// TIA Portal V17 export
// export: Created 2025-03-07T09:16:32.9200456Z, ExportSetting WithDefaults, DisplayName Totally Integrated Automation Portal, DisplayVersion V17 Update 8, DisplayName TIA Portal Openness, DisplayVersion V17 Update 8, DisplayName TIA Portal Version Control Interface, DisplayVersion V17, DisplayName SINAMICS Startdrive Advanced, DisplayVersion V17 SP2, DisplayName SINAMICS Startdrive G110M, G120, G120C, G120D, G120P, G115D, DisplayVersion V17 SP2, DisplayName SINAMICS Startdrive G130, G150, S120, S150, SINAMICS MV, S210, DisplayVersion V17 SP2, DisplayName STEP 7 Professional, DisplayVersion V17 Update 8, DisplayName SINUMERIK ONE STEP 7 Toolbox, DisplayVersion V17 Update 12, DisplayName SINUMERIK 840D sl STEP 7 Toolbox, DisplayVersion V17 Update 12, DisplayName STEP 7 Safety, DisplayVersion V17 Update 6, DisplayName WinCC Advanced, DisplayVersion V17 Update 8
DATA_BLOCK "LBP_SpindleTempSensor"   // DB1002
TITLE = Spindle temperature sensors / Sensores de temperatura del cabezal / Spindeltemperatursensoren
{ S7_Optimized_Access := 'FALSE'; DB_Accessible_From_OPC_UA := 'FALSE' }
AUTHOR : SINUMERIK
FAMILY : SINUMERIK_ONE
VERSION : 6.15
// Interface between user program and operating software, contains signals for spindle temperature sensors / La interfaz entre programa de usuario y software operativo contiene señales para sensores de temperatura del cabezal / Schnittstelle zwischen Anwenderprogramm und Betriebssoftware, enthält Signale für Spindeltemperatursensoren
// stored: AutoNumber false, DBAccessibleFromOPCUA false, DBAccessibleFromWebserver true, IsOnlyStoredInLoadMemory false, IsWriteProtectedInAS false
   VAR RETAIN
      Sp : Array[1..2] of Struct   // Spindel / Spindle / Cabezal
         TS : Array[1..6] of Struct   // Temperatursensor / Temperature sensor / Sensor de temperatura
            MountPlace : Int;   // Platz der Sensorbaugruppe / Sensor assembly location / Ubicación del conjunto de sensores
            Res1 : Int;
            ActVal : Real;   // Temperatursensor Istwert [°C] / Temperature sensor actual value [°C] / Sensor de temperatura valor real [°C]
            WarnThreshold : Real;   // Temperatursensor Warnschwellwert / Temperature sensor warning threshold value [°C] / Sensor de temperatura umbral de alarma
            WarnNumLimitViol : Int;   // Anzahl der Warnschwellwert-Verletzungen / Number of warning threshold value violations / Número de vulneraciones del umbral de alarma
            WarnTsViolYY : Byte;   // Letzte Warnschwellwert-Verletzung: Jahr / Last warning threshold value violation: year / Última vulneración del umbral de alarma: año
            WarnTsViolMM : Byte;   // Letzte Warnschwellwert-Verletzung: Monat / Last warning threshold value violation: month / Última vulneración del umbral de alarma: mes
            WarnTsViolDD : Byte;   // Letzte Warnschwellwert-Verletzung: Tag / Last warning threshold value violation: day / Última vulneración del umbral de fallo: día
            WarnTsViolH : Byte;   // Letzte Warnschwellwert-Verletzung: Stunde / Last warning threshold value violation: hour / Última vulneración del umbral de fallo: hora
            WarnTsViolM : Byte;   // Letzte Warnschwellwert-Verletzung: Minute / Last warning threshold value violation: minute / Última vulneración del umbral de fallo: minuto
            WarnTsViolS : Byte;   // Letzte Warnschwellwert-Verletzung: Sekunde / Last warning threshold value violation: second / Última vulneración del umbral de alarma: segundo
            WarnDurLimitViol : DInt;   // Dauer der Warnschwellwert-Verletzungen / Duration of warning threshold value violations / Duración de vulneraciones del umbral de alarma
            FaultThreshold : Real;   // Temperatursensor Fehlerschwellwert / Temperature sensor fault threshold value [°C] / Sensor de temperatura umbral de fallo
            FaultNumLimitViol : Int;   // Anzahl der Fehlerschwellwert-Verletzungen / Number of fault threshold value violations / Número de vulneraciones del umbral de fallo
            FaultTsViolYY : Byte;   // Letzte Fehlerschwellwert-Verletzung: Jahr / Last fault threshold value violation: year / Última vulneración del umbral de fallo: año
            FaultTsViolMM : Byte;   // Letzte Fehlerschwellwert-Verletzung: Monat / Last fault threshold value violation: month / Última vulneración del umbral de fallo: mes
            FaultTsViolDD : Byte;   // Letzte Fehlerschwellwert-Verletzung: Tag / Last fault threshold value violation: day / Última vulneración del umbral de fallo: día
            FaultTsViolH : Byte;   // Letzte Fehlerschwellwert-Verletzung: Stunde / Last fault threshold value violation: hour / Última vulneración del umbral de fallo: hora
            FaultTsViolM : Byte;   // Letzte Fehlerschwellwert-Verletzung: Minute / Last fault threshold value violation: minute / Última vulneración del umbral de fallo: minuto
            FaultTsViolS : Byte;   // Letzte Fehlerschwellwert-Verletzung: Sekunde / Last fault threshold value violation: second / Última vulneración del umbral de fallo: segundo
            FaultDurLimitViol : DInt;   // Dauer der Fehlerschwellwert-Verletzungen / Duration of fault threshold value violations / Duración de vulneraciones del umbral de fallo
         END_STRUCT;
      END_STRUCT;
   END_VAR
BEGIN
   // Sp[1].TS[2].MountPlace : Platz der Sensorbaugruppe / Sensor assembly location / Ubicación del conjunto de sensores
   // Sp[1].TS[3].MountPlace : Platz der Sensorbaugruppe / Sensor assembly location / Ubicación del conjunto de sensores
   // Sp[1].TS[4].MountPlace : Platz der Sensorbaugruppe / Sensor assembly location / Ubicación del conjunto de sensores
   // Sp[1].TS[5].MountPlace : Platz der Sensorbaugruppe / Sensor assembly location / Ubicación del conjunto de sensores
   // Sp[1].TS[6].MountPlace : Platz der Sensorbaugruppe / Sensor assembly location / Ubicación del conjunto de sensores
   // Sp[2].TS[1].MountPlace : Platz der Sensorbaugruppe / Sensor assembly location / Ubicación del conjunto de sensores
   // Sp[2].TS[2].MountPlace : Platz der Sensorbaugruppe / Sensor assembly location / Ubicación del conjunto de sensores
   // Sp[2].TS[3].MountPlace : Platz der Sensorbaugruppe / Sensor assembly location / Ubicación del conjunto de sensores
   // Sp[2].TS[4].MountPlace : Platz der Sensorbaugruppe / Sensor assembly location / Ubicación del conjunto de sensores
   // Sp[2].TS[5].MountPlace : Platz der Sensorbaugruppe / Sensor assembly location / Ubicación del conjunto de sensores
   // Sp[2].TS[6].MountPlace : Platz der Sensorbaugruppe / Sensor assembly location / Ubicación del conjunto de sensores
   // Sp[1].TS[2].ActVal : Temperatursensor Istwert [°C] / Temperature sensor actual value [°C] / Sensor de temperatura valor real [°C]
   // Sp[1].TS[3].ActVal : Temperatursensor Istwert [°C] / Temperature sensor actual value [°C] / Sensor de temperatura valor real [°C]
   // Sp[1].TS[4].ActVal : Temperatursensor Istwert [°C] / Temperature sensor actual value [°C] / Sensor de temperatura valor real [°C]
   // Sp[1].TS[5].ActVal : Temperatursensor Istwert [°C] / Temperature sensor actual value [°C] / Sensor de temperatura valor real [°C]
   // Sp[1].TS[6].ActVal : Temperatursensor Istwert [°C] / Temperature sensor actual value [°C] / Sensor de temperatura valor real [°C]
   // Sp[2].TS[1].ActVal : Temperatursensor Istwert [°C] / Temperature sensor actual value [°C] / Sensor de temperatura valor real [°C]
   // Sp[2].TS[2].ActVal : Temperatursensor Istwert [°C] / Temperature sensor actual value [°C] / Sensor de temperatura valor real [°C]
   // Sp[2].TS[3].ActVal : Temperatursensor Istwert [°C] / Temperature sensor actual value [°C] / Sensor de temperatura valor real [°C]
   // Sp[2].TS[4].ActVal : Temperatursensor Istwert [°C] / Temperature sensor actual value [°C] / Sensor de temperatura valor real [°C]
   // Sp[2].TS[5].ActVal : Temperatursensor Istwert [°C] / Temperature sensor actual value [°C] / Sensor de temperatura valor real [°C]
   // Sp[2].TS[6].ActVal : Temperatursensor Istwert [°C] / Temperature sensor actual value [°C] / Sensor de temperatura valor real [°C]
   // Sp[1].TS[2].WarnThreshold : Temperatursensor Warnschwellwert / Temperature sensor warning threshold value [°C] / Sensor de temperatura umbral de alarma
   // Sp[1].TS[3].WarnThreshold : Temperatursensor Warnschwellwert / Temperature sensor warning threshold value [°C] / Sensor de temperatura umbral de alarma
   // Sp[1].TS[4].WarnThreshold : Temperatursensor Warnschwellwert / Temperature sensor warning threshold value [°C] / Sensor de temperatura umbral de alarma
   // Sp[1].TS[5].WarnThreshold : Temperatursensor Warnschwellwert / Temperature sensor warning threshold value [°C] / Sensor de temperatura umbral de alarma
   // Sp[1].TS[6].WarnThreshold : Temperatursensor Warnschwellwert / Temperature sensor warning threshold value [°C] / Sensor de temperatura umbral de alarma
   // Sp[2].TS[1].WarnThreshold : Temperatursensor Warnschwellwert / Temperature sensor warning threshold value [°C] / Sensor de temperatura umbral de alarma
   // Sp[2].TS[2].WarnThreshold : Temperatursensor Warnschwellwert / Temperature sensor warning threshold value [°C] / Sensor de temperatura umbral de alarma
   // Sp[2].TS[3].WarnThreshold : Temperatursensor Warnschwellwert / Temperature sensor warning threshold value [°C] / Sensor de temperatura umbral de alarma
   // Sp[2].TS[4].WarnThreshold : Temperatursensor Warnschwellwert / Temperature sensor warning threshold value [°C] / Sensor de temperatura umbral de alarma
   // Sp[2].TS[5].WarnThreshold : Temperatursensor Warnschwellwert / Temperature sensor warning threshold value [°C] / Sensor de temperatura umbral de alarma
   // Sp[2].TS[6].WarnThreshold : Temperatursensor Warnschwellwert / Temperature sensor warning threshold value [°C] / Sensor de temperatura umbral de alarma
   // Sp[1].TS[2].WarnNumLimitViol : Anzahl der Warnschwellwert-Verletzungen / Number of warning threshold value violations / Número de vulneraciones del umbral de alarma
   // Sp[1].TS[3].WarnNumLimitViol : Anzahl der Warnschwellwert-Verletzungen / Number of warning threshold value violations / Número de vulneraciones del umbral de alarma
   // Sp[1].TS[4].WarnNumLimitViol : Anzahl der Warnschwellwert-Verletzungen / Number of warning threshold value violations / Número de vulneraciones del umbral de alarma
   // Sp[1].TS[5].WarnNumLimitViol : Anzahl der Warnschwellwert-Verletzungen / Number of warning threshold value violations / Número de vulneraciones del umbral de alarma
   // Sp[1].TS[6].WarnNumLimitViol : Anzahl der Warnschwellwert-Verletzungen / Number of warning threshold value violations / Número de vulneraciones del umbral de alarma
   // Sp[2].TS[1].WarnNumLimitViol : Anzahl der Warnschwellwert-Verletzungen / Number of warning threshold value violations / Número de vulneraciones del umbral de alarma
   // Sp[2].TS[2].WarnNumLimitViol : Anzahl der Warnschwellwert-Verletzungen / Number of warning threshold value violations / Número de vulneraciones del umbral de alarma
   // Sp[2].TS[3].WarnNumLimitViol : Anzahl der Warnschwellwert-Verletzungen / Number of warning threshold value violations / Número de vulneraciones del umbral de alarma
   // Sp[2].TS[4].WarnNumLimitViol : Anzahl der Warnschwellwert-Verletzungen / Number of warning threshold value violations / Número de vulneraciones del umbral de alarma
   // Sp[2].TS[5].WarnNumLimitViol : Anzahl der Warnschwellwert-Verletzungen / Number of warning threshold value violations / Número de vulneraciones del umbral de alarma
   // Sp[2].TS[6].WarnNumLimitViol : Anzahl der Warnschwellwert-Verletzungen / Number of warning threshold value violations / Número de vulneraciones del umbral de alarma
   // Sp[1].TS[2].WarnTsViolYY : Letzte Warnschwellwert-Verletzung: Jahr / Last warning threshold value violation: year / Última vulneración del umbral de alarma: año
   // Sp[1].TS[3].WarnTsViolYY : Letzte Warnschwellwert-Verletzung: Jahr / Last warning threshold value violation: year / Última vulneración del umbral de alarma: año
   // Sp[1].TS[4].WarnTsViolYY : Letzte Warnschwellwert-Verletzung: Jahr / Last warning threshold value violation: year / Última vulneración del umbral de alarma: año
   // Sp[1].TS[5].WarnTsViolYY : Letzte Warnschwellwert-Verletzung: Jahr / Last warning threshold value violation: year / Última vulneración del umbral de alarma: año
   // Sp[1].TS[6].WarnTsViolYY : Letzte Warnschwellwert-Verletzung: Jahr / Last warning threshold value violation: year / Última vulneración del umbral de alarma: año
   // Sp[2].TS[1].WarnTsViolYY : Letzte Warnschwellwert-Verletzung: Jahr / Last warning threshold value violation: year / Última vulneración del umbral de alarma: año
   // Sp[2].TS[2].WarnTsViolYY : Letzte Warnschwellwert-Verletzung: Jahr / Last warning threshold value violation: year / Última vulneración del umbral de alarma: año
   // Sp[2].TS[3].WarnTsViolYY : Letzte Warnschwellwert-Verletzung: Jahr / Last warning threshold value violation: year / Última vulneración del umbral de alarma: año
   // Sp[2].TS[4].WarnTsViolYY : Letzte Warnschwellwert-Verletzung: Jahr / Last warning threshold value violation: year / Última vulneración del umbral de alarma: año
   // Sp[2].TS[5].WarnTsViolYY : Letzte Warnschwellwert-Verletzung: Jahr / Last warning threshold value violation: year / Última vulneración del umbral de alarma: año
   // Sp[2].TS[6].WarnTsViolYY : Letzte Warnschwellwert-Verletzung: Jahr / Last warning threshold value violation: year / Última vulneración del umbral de alarma: año
   // Sp[1].TS[2].WarnTsViolMM : Letzte Warnschwellwert-Verletzung: Monat / Last warning threshold value violation: month / Última vulneración del umbral de alarma: mes
   // Sp[1].TS[3].WarnTsViolMM : Letzte Warnschwellwert-Verletzung: Monat / Last warning threshold value violation: month / Última vulneración del umbral de alarma: mes
   // Sp[1].TS[4].WarnTsViolMM : Letzte Warnschwellwert-Verletzung: Monat / Last warning threshold value violation: month / Última vulneración del umbral de alarma: mes
   // Sp[1].TS[5].WarnTsViolMM : Letzte Warnschwellwert-Verletzung: Monat / Last warning threshold value violation: month / Última vulneración del umbral de alarma: mes
   // Sp[1].TS[6].WarnTsViolMM : Letzte Warnschwellwert-Verletzung: Monat / Last warning threshold value violation: month / Última vulneración del umbral de alarma: mes
   // Sp[2].TS[1].WarnTsViolMM : Letzte Warnschwellwert-Verletzung: Monat / Last warning threshold value violation: month / Última vulneración del umbral de alarma: mes
   // Sp[2].TS[2].WarnTsViolMM : Letzte Warnschwellwert-Verletzung: Monat / Last warning threshold value violation: month / Última vulneración del umbral de alarma: mes
   // Sp[2].TS[3].WarnTsViolMM : Letzte Warnschwellwert-Verletzung: Monat / Last warning threshold value violation: month / Última vulneración del umbral de alarma: mes
   // Sp[2].TS[4].WarnTsViolMM : Letzte Warnschwellwert-Verletzung: Monat / Last warning threshold value violation: month / Última vulneración del umbral de alarma: mes
   // Sp[2].TS[5].WarnTsViolMM : Letzte Warnschwellwert-Verletzung: Monat / Last warning threshold value violation: month / Última vulneración del umbral de alarma: mes
   // Sp[2].TS[6].WarnTsViolMM : Letzte Warnschwellwert-Verletzung: Monat / Last warning threshold value violation: month / Última vulneración del umbral de alarma: mes
   // Sp[1].TS[2].WarnTsViolDD : Letzte Warnschwellwert-Verletzung: Tag / Last warning threshold value violation: day / Última vulneración del umbral de fallo: día
   // Sp[1].TS[3].WarnTsViolDD : Letzte Warnschwellwert-Verletzung: Tag / Last warning threshold value violation: day / Última vulneración del umbral de fallo: día
   // Sp[1].TS[4].WarnTsViolDD : Letzte Warnschwellwert-Verletzung: Tag / Last warning threshold value violation: day / Última vulneración del umbral de fallo: día
   // Sp[1].TS[5].WarnTsViolDD : Letzte Warnschwellwert-Verletzung: Tag / Last warning threshold value violation: day / Última vulneración del umbral de fallo: día
   // Sp[1].TS[6].WarnTsViolDD : Letzte Warnschwellwert-Verletzung: Tag / Last warning threshold value violation: day / Última vulneración del umbral de fallo: día
   // Sp[2].TS[1].WarnTsViolDD : Letzte Warnschwellwert-Verletzung: Tag / Last warning threshold value violation: day / Última vulneración del umbral de fallo: día
   // Sp[2].TS[2].WarnTsViolDD : Letzte Warnschwellwert-Verletzung: Tag / Last warning threshold value violation: day / Última vulneración del umbral de fallo: día
   // Sp[2].TS[3].WarnTsViolDD : Letzte Warnschwellwert-Verletzung: Tag / Last warning threshold value violation: day / Última vulneración del umbral de fallo: día
   // Sp[2].TS[4].WarnTsViolDD : Letzte Warnschwellwert-Verletzung: Tag / Last warning threshold value violation: day / Última vulneración del umbral de fallo: día
   // Sp[2].TS[5].WarnTsViolDD : Letzte Warnschwellwert-Verletzung: Tag / Last warning threshold value violation: day / Última vulneración del umbral de fallo: día
   // Sp[2].TS[6].WarnTsViolDD : Letzte Warnschwellwert-Verletzung: Tag / Last warning threshold value violation: day / Última vulneración del umbral de fallo: día
   // Sp[1].TS[2].WarnTsViolH : Letzte Warnschwellwert-Verletzung: Stunde / Last warning threshold value violation: hour / Última vulneración del umbral de fallo: hora
   // Sp[1].TS[3].WarnTsViolH : Letzte Warnschwellwert-Verletzung: Stunde / Last warning threshold value violation: hour / Última vulneración del umbral de fallo: hora
   // Sp[1].TS[4].WarnTsViolH : Letzte Warnschwellwert-Verletzung: Stunde / Last warning threshold value violation: hour / Última vulneración del umbral de fallo: hora
   // Sp[1].TS[5].WarnTsViolH : Letzte Warnschwellwert-Verletzung: Stunde / Last warning threshold value violation: hour / Última vulneración del umbral de fallo: hora
   // Sp[1].TS[6].WarnTsViolH : Letzte Warnschwellwert-Verletzung: Stunde / Last warning threshold value violation: hour / Última vulneración del umbral de fallo: hora
   // Sp[2].TS[1].WarnTsViolH : Letzte Warnschwellwert-Verletzung: Stunde / Last warning threshold value violation: hour / Última vulneración del umbral de fallo: hora
   // Sp[2].TS[2].WarnTsViolH : Letzte Warnschwellwert-Verletzung: Stunde / Last warning threshold value violation: hour / Última vulneración del umbral de fallo: hora
   // Sp[2].TS[3].WarnTsViolH : Letzte Warnschwellwert-Verletzung: Stunde / Last warning threshold value violation: hour / Última vulneración del umbral de fallo: hora
   // Sp[2].TS[4].WarnTsViolH : Letzte Warnschwellwert-Verletzung: Stunde / Last warning threshold value violation: hour / Última vulneración del umbral de fallo: hora
   // Sp[2].TS[5].WarnTsViolH : Letzte Warnschwellwert-Verletzung: Stunde / Last warning threshold value violation: hour / Última vulneración del umbral de fallo: hora
   // Sp[2].TS[6].WarnTsViolH : Letzte Warnschwellwert-Verletzung: Stunde / Last warning threshold value violation: hour / Última vulneración del umbral de fallo: hora
   // Sp[1].TS[2].WarnTsViolM : Letzte Warnschwellwert-Verletzung: Minute / Last warning threshold value violation: minute / Última vulneración del umbral de fallo: minuto
   // Sp[1].TS[3].WarnTsViolM : Letzte Warnschwellwert-Verletzung: Minute / Last warning threshold value violation: minute / Última vulneración del umbral de fallo: minuto
   // Sp[1].TS[4].WarnTsViolM : Letzte Warnschwellwert-Verletzung: Minute / Last warning threshold value violation: minute / Última vulneración del umbral de fallo: minuto
   // Sp[1].TS[5].WarnTsViolM : Letzte Warnschwellwert-Verletzung: Minute / Last warning threshold value violation: minute / Última vulneración del umbral de fallo: minuto
   // Sp[1].TS[6].WarnTsViolM : Letzte Warnschwellwert-Verletzung: Minute / Last warning threshold value violation: minute / Última vulneración del umbral de fallo: minuto
   // Sp[2].TS[1].WarnTsViolM : Letzte Warnschwellwert-Verletzung: Minute / Last warning threshold value violation: minute / Última vulneración del umbral de fallo: minuto
   // Sp[2].TS[2].WarnTsViolM : Letzte Warnschwellwert-Verletzung: Minute / Last warning threshold value violation: minute / Última vulneración del umbral de fallo: minuto
   // Sp[2].TS[3].WarnTsViolM : Letzte Warnschwellwert-Verletzung: Minute / Last warning threshold value violation: minute / Última vulneración del umbral de fallo: minuto
   // Sp[2].TS[4].WarnTsViolM : Letzte Warnschwellwert-Verletzung: Minute / Last warning threshold value violation: minute / Última vulneración del umbral de fallo: minuto
   // Sp[2].TS[5].WarnTsViolM : Letzte Warnschwellwert-Verletzung: Minute / Last warning threshold value violation: minute / Última vulneración del umbral de fallo: minuto
   // Sp[2].TS[6].WarnTsViolM : Letzte Warnschwellwert-Verletzung: Minute / Last warning threshold value violation: minute / Última vulneración del umbral de fallo: minuto
   // Sp[1].TS[2].WarnTsViolS : Letzte Warnschwellwert-Verletzung: Sekunde / Last warning threshold value violation: second / Última vulneración del umbral de alarma: segundo
   // Sp[1].TS[3].WarnTsViolS : Letzte Warnschwellwert-Verletzung: Sekunde / Last warning threshold value violation: second / Última vulneración del umbral de alarma: segundo
   // Sp[1].TS[4].WarnTsViolS : Letzte Warnschwellwert-Verletzung: Sekunde / Last warning threshold value violation: second / Última vulneración del umbral de alarma: segundo
   // Sp[1].TS[5].WarnTsViolS : Letzte Warnschwellwert-Verletzung: Sekunde / Last warning threshold value violation: second / Última vulneración del umbral de alarma: segundo
   // Sp[1].TS[6].WarnTsViolS : Letzte Warnschwellwert-Verletzung: Sekunde / Last warning threshold value violation: second / Última vulneración del umbral de alarma: segundo
   // Sp[2].TS[1].WarnTsViolS : Letzte Warnschwellwert-Verletzung: Sekunde / Last warning threshold value violation: second / Última vulneración del umbral de alarma: segundo
   // Sp[2].TS[2].WarnTsViolS : Letzte Warnschwellwert-Verletzung: Sekunde / Last warning threshold value violation: second / Última vulneración del umbral de alarma: segundo
   // Sp[2].TS[3].WarnTsViolS : Letzte Warnschwellwert-Verletzung: Sekunde / Last warning threshold value violation: second / Última vulneración del umbral de alarma: segundo
   // Sp[2].TS[4].WarnTsViolS : Letzte Warnschwellwert-Verletzung: Sekunde / Last warning threshold value violation: second / Última vulneración del umbral de alarma: segundo
   // Sp[2].TS[5].WarnTsViolS : Letzte Warnschwellwert-Verletzung: Sekunde / Last warning threshold value violation: second / Última vulneración del umbral de alarma: segundo
   // Sp[2].TS[6].WarnTsViolS : Letzte Warnschwellwert-Verletzung: Sekunde / Last warning threshold value violation: second / Última vulneración del umbral de alarma: segundo
   // Sp[1].TS[2].WarnDurLimitViol : Dauer der Warnschwellwert-Verletzungen / Duration of warning threshold value violations / Duración de vulneraciones del umbral de alarma
   // Sp[1].TS[3].WarnDurLimitViol : Dauer der Warnschwellwert-Verletzungen / Duration of warning threshold value violations / Duración de vulneraciones del umbral de alarma
   // Sp[1].TS[4].WarnDurLimitViol : Dauer der Warnschwellwert-Verletzungen / Duration of warning threshold value violations / Duración de vulneraciones del umbral de alarma
   // Sp[1].TS[5].WarnDurLimitViol : Dauer der Warnschwellwert-Verletzungen / Duration of warning threshold value violations / Duración de vulneraciones del umbral de alarma
   // Sp[1].TS[6].WarnDurLimitViol : Dauer der Warnschwellwert-Verletzungen / Duration of warning threshold value violations / Duración de vulneraciones del umbral de alarma
   // Sp[2].TS[1].WarnDurLimitViol : Dauer der Warnschwellwert-Verletzungen / Duration of warning threshold value violations / Duración de vulneraciones del umbral de alarma
   // Sp[2].TS[2].WarnDurLimitViol : Dauer der Warnschwellwert-Verletzungen / Duration of warning threshold value violations / Duración de vulneraciones del umbral de alarma
   // Sp[2].TS[3].WarnDurLimitViol : Dauer der Warnschwellwert-Verletzungen / Duration of warning threshold value violations / Duración de vulneraciones del umbral de alarma
   // Sp[2].TS[4].WarnDurLimitViol : Dauer der Warnschwellwert-Verletzungen / Duration of warning threshold value violations / Duración de vulneraciones del umbral de alarma
   // Sp[2].TS[5].WarnDurLimitViol : Dauer der Warnschwellwert-Verletzungen / Duration of warning threshold value violations / Duración de vulneraciones del umbral de alarma
   // Sp[2].TS[6].WarnDurLimitViol : Dauer der Warnschwellwert-Verletzungen / Duration of warning threshold value violations / Duración de vulneraciones del umbral de alarma
   // Sp[1].TS[2].FaultThreshold : Temperatursensor Fehlerschwellwert / Temperature sensor fault threshold value [°C] / Sensor de temperatura umbral de fallo
   // Sp[1].TS[3].FaultThreshold : Temperatursensor Fehlerschwellwert / Temperature sensor fault threshold value [°C] / Sensor de temperatura umbral de fallo
   // Sp[1].TS[4].FaultThreshold : Temperatursensor Fehlerschwellwert / Temperature sensor fault threshold value [°C] / Sensor de temperatura umbral de fallo
   // Sp[1].TS[5].FaultThreshold : Temperatursensor Fehlerschwellwert / Temperature sensor fault threshold value [°C] / Sensor de temperatura umbral de fallo
   // Sp[1].TS[6].FaultThreshold : Temperatursensor Fehlerschwellwert / Temperature sensor fault threshold value [°C] / Sensor de temperatura umbral de fallo
   // Sp[2].TS[1].FaultThreshold : Temperatursensor Fehlerschwellwert / Temperature sensor fault threshold value [°C] / Sensor de temperatura umbral de fallo
   // Sp[2].TS[2].FaultThreshold : Temperatursensor Fehlerschwellwert / Temperature sensor fault threshold value [°C] / Sensor de temperatura umbral de fallo
   // Sp[2].TS[3].FaultThreshold : Temperatursensor Fehlerschwellwert / Temperature sensor fault threshold value [°C] / Sensor de temperatura umbral de fallo
   // Sp[2].TS[4].FaultThreshold : Temperatursensor Fehlerschwellwert / Temperature sensor fault threshold value [°C] / Sensor de temperatura umbral de fallo
   // Sp[2].TS[5].FaultThreshold : Temperatursensor Fehlerschwellwert / Temperature sensor fault threshold value [°C] / Sensor de temperatura umbral de fallo
   // Sp[2].TS[6].FaultThreshold : Temperatursensor Fehlerschwellwert / Temperature sensor fault threshold value [°C] / Sensor de temperatura umbral de fallo
   // Sp[1].TS[2].FaultNumLimitViol : Anzahl der Fehlerschwellwert-Verletzungen / Number of fault threshold value violations / Número de vulneraciones del umbral de fallo
   // Sp[1].TS[3].FaultNumLimitViol : Anzahl der Fehlerschwellwert-Verletzungen / Number of fault threshold value violations / Número de vulneraciones del umbral de fallo
   // Sp[1].TS[4].FaultNumLimitViol : Anzahl der Fehlerschwellwert-Verletzungen / Number of fault threshold value violations / Número de vulneraciones del umbral de fallo
   // Sp[1].TS[5].FaultNumLimitViol : Anzahl der Fehlerschwellwert-Verletzungen / Number of fault threshold value violations / Número de vulneraciones del umbral de fallo
   // Sp[1].TS[6].FaultNumLimitViol : Anzahl der Fehlerschwellwert-Verletzungen / Number of fault threshold value violations / Número de vulneraciones del umbral de fallo
   // Sp[2].TS[1].FaultNumLimitViol : Anzahl der Fehlerschwellwert-Verletzungen / Number of fault threshold value violations / Número de vulneraciones del umbral de fallo
   // Sp[2].TS[2].FaultNumLimitViol : Anzahl der Fehlerschwellwert-Verletzungen / Number of fault threshold value violations / Número de vulneraciones del umbral de fallo
   // Sp[2].TS[3].FaultNumLimitViol : Anzahl der Fehlerschwellwert-Verletzungen / Number of fault threshold value violations / Número de vulneraciones del umbral de fallo
   // Sp[2].TS[4].FaultNumLimitViol : Anzahl der Fehlerschwellwert-Verletzungen / Number of fault threshold value violations / Número de vulneraciones del umbral de fallo
   // Sp[2].TS[5].FaultNumLimitViol : Anzahl der Fehlerschwellwert-Verletzungen / Number of fault threshold value violations / Número de vulneraciones del umbral de fallo
   // Sp[2].TS[6].FaultNumLimitViol : Anzahl der Fehlerschwellwert-Verletzungen / Number of fault threshold value violations / Número de vulneraciones del umbral de fallo
   // Sp[1].TS[2].FaultTsViolYY : Letzte Fehlerschwellwert-Verletzung: Jahr / Last fault threshold value violation: year / Última vulneración del umbral de fallo: año
   // Sp[1].TS[3].FaultTsViolYY : Letzte Fehlerschwellwert-Verletzung: Jahr / Last fault threshold value violation: year / Última vulneración del umbral de fallo: año
   // Sp[1].TS[4].FaultTsViolYY : Letzte Fehlerschwellwert-Verletzung: Jahr / Last fault threshold value violation: year / Última vulneración del umbral de fallo: año
   // Sp[1].TS[5].FaultTsViolYY : Letzte Fehlerschwellwert-Verletzung: Jahr / Last fault threshold value violation: year / Última vulneración del umbral de fallo: año
   // Sp[1].TS[6].FaultTsViolYY : Letzte Fehlerschwellwert-Verletzung: Jahr / Last fault threshold value violation: year / Última vulneración del umbral de fallo: año
   // Sp[2].TS[1].FaultTsViolYY : Letzte Fehlerschwellwert-Verletzung: Jahr / Last fault threshold value violation: year / Última vulneración del umbral de fallo: año
   // Sp[2].TS[2].FaultTsViolYY : Letzte Fehlerschwellwert-Verletzung: Jahr / Last fault threshold value violation: year / Última vulneración del umbral de fallo: año
   // Sp[2].TS[3].FaultTsViolYY : Letzte Fehlerschwellwert-Verletzung: Jahr / Last fault threshold value violation: year / Última vulneración del umbral de fallo: año
   // Sp[2].TS[4].FaultTsViolYY : Letzte Fehlerschwellwert-Verletzung: Jahr / Last fault threshold value violation: year / Última vulneración del umbral de fallo: año
   // Sp[2].TS[5].FaultTsViolYY : Letzte Fehlerschwellwert-Verletzung: Jahr / Last fault threshold value violation: year / Última vulneración del umbral de fallo: año
   // Sp[2].TS[6].FaultTsViolYY : Letzte Fehlerschwellwert-Verletzung: Jahr / Last fault threshold value violation: year / Última vulneración del umbral de fallo: año
   // Sp[1].TS[2].FaultTsViolMM : Letzte Fehlerschwellwert-Verletzung: Monat / Last fault threshold value violation: month / Última vulneración del umbral de fallo: mes
   // Sp[1].TS[3].FaultTsViolMM : Letzte Fehlerschwellwert-Verletzung: Monat / Last fault threshold value violation: month / Última vulneración del umbral de fallo: mes
   // Sp[1].TS[4].FaultTsViolMM : Letzte Fehlerschwellwert-Verletzung: Monat / Last fault threshold value violation: month / Última vulneración del umbral de fallo: mes
   // Sp[1].TS[5].FaultTsViolMM : Letzte Fehlerschwellwert-Verletzung: Monat / Last fault threshold value violation: month / Última vulneración del umbral de fallo: mes
   // Sp[1].TS[6].FaultTsViolMM : Letzte Fehlerschwellwert-Verletzung: Monat / Last fault threshold value violation: month / Última vulneración del umbral de fallo: mes
   // Sp[2].TS[1].FaultTsViolMM : Letzte Fehlerschwellwert-Verletzung: Monat / Last fault threshold value violation: month / Última vulneración del umbral de fallo: mes
   // Sp[2].TS[2].FaultTsViolMM : Letzte Fehlerschwellwert-Verletzung: Monat / Last fault threshold value violation: month / Última vulneración del umbral de fallo: mes
   // Sp[2].TS[3].FaultTsViolMM : Letzte Fehlerschwellwert-Verletzung: Monat / Last fault threshold value violation: month / Última vulneración del umbral de fallo: mes
   // Sp[2].TS[4].FaultTsViolMM : Letzte Fehlerschwellwert-Verletzung: Monat / Last fault threshold value violation: month / Última vulneración del umbral de fallo: mes
   // Sp[2].TS[5].FaultTsViolMM : Letzte Fehlerschwellwert-Verletzung: Monat / Last fault threshold value violation: month / Última vulneración del umbral de fallo: mes
   // Sp[2].TS[6].FaultTsViolMM : Letzte Fehlerschwellwert-Verletzung: Monat / Last fault threshold value violation: month / Última vulneración del umbral de fallo: mes
   // Sp[1].TS[2].FaultTsViolDD : Letzte Fehlerschwellwert-Verletzung: Tag / Last fault threshold value violation: day / Última vulneración del umbral de fallo: día
   // Sp[1].TS[3].FaultTsViolDD : Letzte Fehlerschwellwert-Verletzung: Tag / Last fault threshold value violation: day / Última vulneración del umbral de fallo: día
   // Sp[1].TS[4].FaultTsViolDD : Letzte Fehlerschwellwert-Verletzung: Tag / Last fault threshold value violation: day / Última vulneración del umbral de fallo: día
   // Sp[1].TS[5].FaultTsViolDD : Letzte Fehlerschwellwert-Verletzung: Tag / Last fault threshold value violation: day / Última vulneración del umbral de fallo: día
   // Sp[1].TS[6].FaultTsViolDD : Letzte Fehlerschwellwert-Verletzung: Tag / Last fault threshold value violation: day / Última vulneración del umbral de fallo: día
   // Sp[2].TS[1].FaultTsViolDD : Letzte Fehlerschwellwert-Verletzung: Tag / Last fault threshold value violation: day / Última vulneración del umbral de fallo: día
   // Sp[2].TS[2].FaultTsViolDD : Letzte Fehlerschwellwert-Verletzung: Tag / Last fault threshold value violation: day / Última vulneración del umbral de fallo: día
   // Sp[2].TS[3].FaultTsViolDD : Letzte Fehlerschwellwert-Verletzung: Tag / Last fault threshold value violation: day / Última vulneración del umbral de fallo: día
   // Sp[2].TS[4].FaultTsViolDD : Letzte Fehlerschwellwert-Verletzung: Tag / Last fault threshold value violation: day / Última vulneración del umbral de fallo: día
   // Sp[2].TS[5].FaultTsViolDD : Letzte Fehlerschwellwert-Verletzung: Tag / Last fault threshold value violation: day / Última vulneración del umbral de fallo: día
   // Sp[2].TS[6].FaultTsViolDD : Letzte Fehlerschwellwert-Verletzung: Tag / Last fault threshold value violation: day / Última vulneración del umbral de fallo: día
   // Sp[1].TS[2].FaultTsViolH : Letzte Fehlerschwellwert-Verletzung: Stunde / Last fault threshold value violation: hour / Última vulneración del umbral de fallo: hora
   // Sp[1].TS[3].FaultTsViolH : Letzte Fehlerschwellwert-Verletzung: Stunde / Last fault threshold value violation: hour / Última vulneración del umbral de fallo: hora
   // Sp[1].TS[4].FaultTsViolH : Letzte Fehlerschwellwert-Verletzung: Stunde / Last fault threshold value violation: hour / Última vulneración del umbral de fallo: hora
   // Sp[1].TS[5].FaultTsViolH : Letzte Fehlerschwellwert-Verletzung: Stunde / Last fault threshold value violation: hour / Última vulneración del umbral de fallo: hora
   // Sp[1].TS[6].FaultTsViolH : Letzte Fehlerschwellwert-Verletzung: Stunde / Last fault threshold value violation: hour / Última vulneración del umbral de fallo: hora
   // Sp[2].TS[1].FaultTsViolH : Letzte Fehlerschwellwert-Verletzung: Stunde / Last fault threshold value violation: hour / Última vulneración del umbral de fallo: hora
   // Sp[2].TS[2].FaultTsViolH : Letzte Fehlerschwellwert-Verletzung: Stunde / Last fault threshold value violation: hour / Última vulneración del umbral de fallo: hora
   // Sp[2].TS[3].FaultTsViolH : Letzte Fehlerschwellwert-Verletzung: Stunde / Last fault threshold value violation: hour / Última vulneración del umbral de fallo: hora
   // Sp[2].TS[4].FaultTsViolH : Letzte Fehlerschwellwert-Verletzung: Stunde / Last fault threshold value violation: hour / Última vulneración del umbral de fallo: hora
   // Sp[2].TS[5].FaultTsViolH : Letzte Fehlerschwellwert-Verletzung: Stunde / Last fault threshold value violation: hour / Última vulneración del umbral de fallo: hora
   // Sp[2].TS[6].FaultTsViolH : Letzte Fehlerschwellwert-Verletzung: Stunde / Last fault threshold value violation: hour / Última vulneración del umbral de fallo: hora
   // Sp[1].TS[2].FaultTsViolM : Letzte Fehlerschwellwert-Verletzung: Minute / Last fault threshold value violation: minute / Última vulneración del umbral de fallo: minuto
   // Sp[1].TS[3].FaultTsViolM : Letzte Fehlerschwellwert-Verletzung: Minute / Last fault threshold value violation: minute / Última vulneración del umbral de fallo: minuto
   // Sp[1].TS[4].FaultTsViolM : Letzte Fehlerschwellwert-Verletzung: Minute / Last fault threshold value violation: minute / Última vulneración del umbral de fallo: minuto
   // Sp[1].TS[5].FaultTsViolM : Letzte Fehlerschwellwert-Verletzung: Minute / Last fault threshold value violation: minute / Última vulneración del umbral de fallo: minuto
   // Sp[1].TS[6].FaultTsViolM : Letzte Fehlerschwellwert-Verletzung: Minute / Last fault threshold value violation: minute / Última vulneración del umbral de fallo: minuto
   // Sp[2].TS[1].FaultTsViolM : Letzte Fehlerschwellwert-Verletzung: Minute / Last fault threshold value violation: minute / Última vulneración del umbral de fallo: minuto
   // Sp[2].TS[2].FaultTsViolM : Letzte Fehlerschwellwert-Verletzung: Minute / Last fault threshold value violation: minute / Última vulneración del umbral de fallo: minuto
   // Sp[2].TS[3].FaultTsViolM : Letzte Fehlerschwellwert-Verletzung: Minute / Last fault threshold value violation: minute / Última vulneración del umbral de fallo: minuto
   // Sp[2].TS[4].FaultTsViolM : Letzte Fehlerschwellwert-Verletzung: Minute / Last fault threshold value violation: minute / Última vulneración del umbral de fallo: minuto
   // Sp[2].TS[5].FaultTsViolM : Letzte Fehlerschwellwert-Verletzung: Minute / Last fault threshold value violation: minute / Última vulneración del umbral de fallo: minuto
   // Sp[2].TS[6].FaultTsViolM : Letzte Fehlerschwellwert-Verletzung: Minute / Last fault threshold value violation: minute / Última vulneración del umbral de fallo: minuto
   // Sp[1].TS[2].FaultTsViolS : Letzte Fehlerschwellwert-Verletzung: Sekunde / Last fault threshold value violation: second / Última vulneración del umbral de fallo: segundo
   // Sp[1].TS[3].FaultTsViolS : Letzte Fehlerschwellwert-Verletzung: Sekunde / Last fault threshold value violation: second / Última vulneración del umbral de fallo: segundo
   // Sp[1].TS[4].FaultTsViolS : Letzte Fehlerschwellwert-Verletzung: Sekunde / Last fault threshold value violation: second / Última vulneración del umbral de fallo: segundo
   // Sp[1].TS[5].FaultTsViolS : Letzte Fehlerschwellwert-Verletzung: Sekunde / Last fault threshold value violation: second / Última vulneración del umbral de fallo: segundo
   // Sp[1].TS[6].FaultTsViolS : Letzte Fehlerschwellwert-Verletzung: Sekunde / Last fault threshold value violation: second / Última vulneración del umbral de fallo: segundo
   // Sp[2].TS[1].FaultTsViolS : Letzte Fehlerschwellwert-Verletzung: Sekunde / Last fault threshold value violation: second / Última vulneración del umbral de fallo: segundo
   // Sp[2].TS[2].FaultTsViolS : Letzte Fehlerschwellwert-Verletzung: Sekunde / Last fault threshold value violation: second / Última vulneración del umbral de fallo: segundo
   // Sp[2].TS[3].FaultTsViolS : Letzte Fehlerschwellwert-Verletzung: Sekunde / Last fault threshold value violation: second / Última vulneración del umbral de fallo: segundo
   // Sp[2].TS[4].FaultTsViolS : Letzte Fehlerschwellwert-Verletzung: Sekunde / Last fault threshold value violation: second / Última vulneración del umbral de fallo: segundo
   // Sp[2].TS[5].FaultTsViolS : Letzte Fehlerschwellwert-Verletzung: Sekunde / Last fault threshold value violation: second / Última vulneración del umbral de fallo: segundo
   // Sp[2].TS[6].FaultTsViolS : Letzte Fehlerschwellwert-Verletzung: Sekunde / Last fault threshold value violation: second / Última vulneración del umbral de fallo: segundo
   // Sp[1].TS[2].FaultDurLimitViol : Dauer der Fehlerschwellwert-Verletzungen / Duration of fault threshold value violations / Duración de vulneraciones del umbral de fallo
   // Sp[1].TS[3].FaultDurLimitViol : Dauer der Fehlerschwellwert-Verletzungen / Duration of fault threshold value violations / Duración de vulneraciones del umbral de fallo
   // Sp[1].TS[4].FaultDurLimitViol : Dauer der Fehlerschwellwert-Verletzungen / Duration of fault threshold value violations / Duración de vulneraciones del umbral de fallo
   // Sp[1].TS[5].FaultDurLimitViol : Dauer der Fehlerschwellwert-Verletzungen / Duration of fault threshold value violations / Duración de vulneraciones del umbral de fallo
   // Sp[1].TS[6].FaultDurLimitViol : Dauer der Fehlerschwellwert-Verletzungen / Duration of fault threshold value violations / Duración de vulneraciones del umbral de fallo
   // Sp[2].TS[1].FaultDurLimitViol : Dauer der Fehlerschwellwert-Verletzungen / Duration of fault threshold value violations / Duración de vulneraciones del umbral de fallo
   // Sp[2].TS[2].FaultDurLimitViol : Dauer der Fehlerschwellwert-Verletzungen / Duration of fault threshold value violations / Duración de vulneraciones del umbral de fallo
   // Sp[2].TS[3].FaultDurLimitViol : Dauer der Fehlerschwellwert-Verletzungen / Duration of fault threshold value violations / Duración de vulneraciones del umbral de fallo
   // Sp[2].TS[4].FaultDurLimitViol : Dauer der Fehlerschwellwert-Verletzungen / Duration of fault threshold value violations / Duración de vulneraciones del umbral de fallo
   // Sp[2].TS[5].FaultDurLimitViol : Dauer der Fehlerschwellwert-Verletzungen / Duration of fault threshold value violations / Duración de vulneraciones del umbral de fallo
   // Sp[2].TS[6].FaultDurLimitViol : Dauer der Fehlerschwellwert-Verletzungen / Duration of fault threshold value violations / Duración de vulneraciones del umbral de fallo
   // Sp[1].TS[1] : Temperatursensor / Temperature sensor / Sensor de temperatura
   // Sp[1].TS[2] : Temperatursensor / Temperature sensor / Sensor de temperatura
   // Sp[1].TS[3] : Temperatursensor / Temperature sensor / Sensor de temperatura
   // Sp[1].TS[4] : Temperatursensor / Temperature sensor / Sensor de temperatura
   // Sp[1].TS[5] : Temperatursensor / Temperature sensor / Sensor de temperatura
   // Sp[1].TS[6] : Temperatursensor / Temperature sensor / Sensor de temperatura
   // Sp[2].TS[1] : Temperatursensor / Temperature sensor / Sensor de temperatura
   // Sp[2].TS[2] : Temperatursensor / Temperature sensor / Sensor de temperatura
   // Sp[2].TS[3] : Temperatursensor / Temperature sensor / Sensor de temperatura
   // Sp[2].TS[4] : Temperatursensor / Temperature sensor / Sensor de temperatura
   // Sp[2].TS[5] : Temperatursensor / Temperature sensor / Sensor de temperatura
   // Sp[2].TS[6] : Temperatursensor / Temperature sensor / Sensor de temperatura
   // Sp[2].TS : Temperatursensor / Temperature sensor / Sensor de temperatura
   // Sp[1] : Spindel / Spindle / Cabezal
   // Sp[2] : Spindel / Spindle / Cabezal
END_DATA_BLOCK
